_CFC_ (* Continuous Function Chart, elements in execution order *)
#0 ABS(SCHU_P2_2_YA3_RASSOG)
#1 GT(#0, SCHU_P2_2_YA3_UST_RAS_TEMP)
#2 ABS(SCHU_P2_2_YA3_RASSOG_POL)
#3 GT(#2, SCHU_P2_2_YA3_UST_RAS_POL)
#4 OR(#1, #3)
#5 AND(SCHU_P2_2_UST_LETO, SCHU_P2_2_UST_RE_RABOTA, #4)
#6 INT_TO_TIME(SCHU_P2_2_YA3_ZADER_OTK)
#7 MUL(#6, 1000)
#8 TON_YA3_Zakl:TON(IN: #5, PT: #7)
#9 OR(#8.Q, YA3_AO_OTKAZ, YA3_OTKAZ)
#10 AND(SCHU_P2_2_UE2_T_DOST, SCHU_P2_2_SA5_DI5_A, #9)
#11 SR_YA3_Otk:SR(SET1: #10, RESET: SCHU_P2_2_SB)
#12 SCHU_P2_2_Z_YA3_OTKAZ <= #11.Q1
_END_CFC_
(* the same logic as Structured Text *)
TON_YA3_Zakl(IN := SCHU_P2_2_UST_LETO AND SCHU_P2_2_UST_RE_RABOTA AND ((ABS(SCHU_P2_2_YA3_RASSOG) > SCHU_P2_2_YA3_UST_RAS_TEMP) OR (ABS(SCHU_P2_2_YA3_RASSOG_POL) > SCHU_P2_2_YA3_UST_RAS_POL)), PT := INT_TO_TIME(SCHU_P2_2_YA3_ZADER_OTK) * 1000);
SR_YA3_Otk(SET1 := SCHU_P2_2_UE2_T_DOST AND SCHU_P2_2_SA5_DI5_A AND (TON_YA3_Zakl.Q OR YA3_AO_OTKAZ OR YA3_OTKAZ), RESET := SCHU_P2_2_SB);
SCHU_P2_2_Z_YA3_OTKAZ := SR_YA3_Otk.Q1;
END_PROGRAM

(* POU TZBiS/TZB/Z_YA4_Otk, CFC *)
PROGRAM Z_YA4_Otk
VAR
	RS_YA4_OTKZ: SR;

	UE3_ZADER: TON;
	SCHU_P2_2_YA4_AO4ER: TON;
	F_trig_ai: F_TRIG;
	TON_YA4: TON;
	YA4_ZADER_POL: TON;
	YA4_ZADER_TEMP: TON;
END_VAR
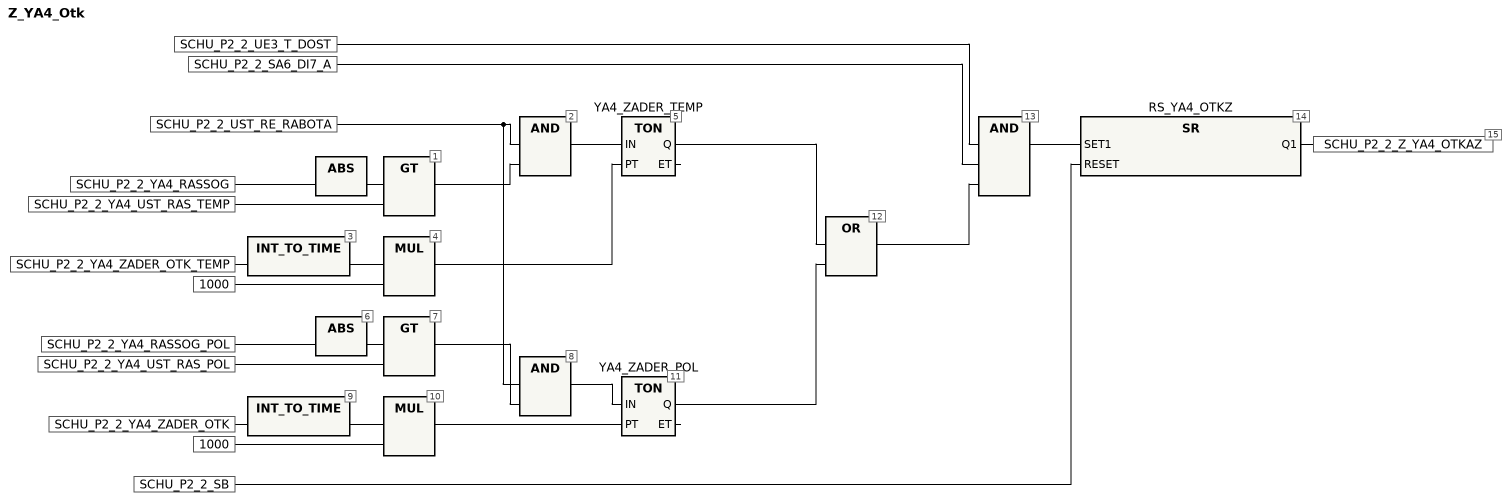
_CFC_ (* Continuous Function Chart, elements in execution order *)
#0 ABS(SCHU_P2_2_YA4_RASSOG)
#1 GT(#0, SCHU_P2_2_YA4_UST_RAS_TEMP)
#2 AND(SCHU_P2_2_UST_RE_RABOTA, #1)
#3 INT_TO_TIME(SCHU_P2_2_YA4_ZADER_OTK_TEMP)
#4 MUL(#3, 1000)
#5 YA4_ZADER_TEMP:TON(IN: #2, PT: #4)
#6 ABS(SCHU_P2_2_YA4_RASSOG_POL)
#7 GT(#6, SCHU_P2_2_YA4_UST_RAS_POL)
#8 AND(SCHU_P2_2_UST_RE_RABOTA, #7)
#9 INT_TO_TIME(SCHU_P2_2_YA4_ZADER_OTK)
#10 MUL(#9, 1000)
#11 YA4_ZADER_POL:TON(IN: #8, PT: #10)
#12 OR(#5.Q, #11.Q)
#13 AND(SCHU_P2_2_UE3_T_DOST, SCHU_P2_2_SA6_DI7_A, #12)
#14 RS_YA4_OTKZ:SR(SET1: #13, RESET: SCHU_P2_2_SB)
#15 SCHU_P2_2_Z_YA4_OTKAZ <= #14.Q1
_END_CFC_
(* the same logic as Structured Text *)
YA4_ZADER_TEMP(IN := SCHU_P2_2_UST_RE_RABOTA AND (ABS(SCHU_P2_2_YA4_RASSOG) > SCHU_P2_2_YA4_UST_RAS_TEMP), PT := INT_TO_TIME(SCHU_P2_2_YA4_ZADER_OTK_TEMP) * 1000);
YA4_ZADER_POL(IN := SCHU_P2_2_UST_RE_RABOTA AND (ABS(SCHU_P2_2_YA4_RASSOG_POL) > SCHU_P2_2_YA4_UST_RAS_POL), PT := INT_TO_TIME(SCHU_P2_2_YA4_ZADER_OTK) * 1000);
RS_YA4_OTKZ(SET1 := SCHU_P2_2_UE3_T_DOST AND SCHU_P2_2_SA6_DI7_A AND (YA4_ZADER_TEMP.Q OR YA4_ZADER_POL.Q), RESET := SCHU_P2_2_SB);
SCHU_P2_2_Z_YA4_OTKAZ := RS_YA4_OTKZ.Q1;
END_PROGRAM

(* POU TZBiS/TZB/Z_Zam, CFC *)
PROGRAM Z_Zam
VAR
	RT_VKL: R_TRIG;
	SR_ZAM: SR;
	TON_VKL: TON;
	TP_VKL: TON;
	FT_TP_VKL: F_TRIG;
	SR_TS: SR;
END_VAR
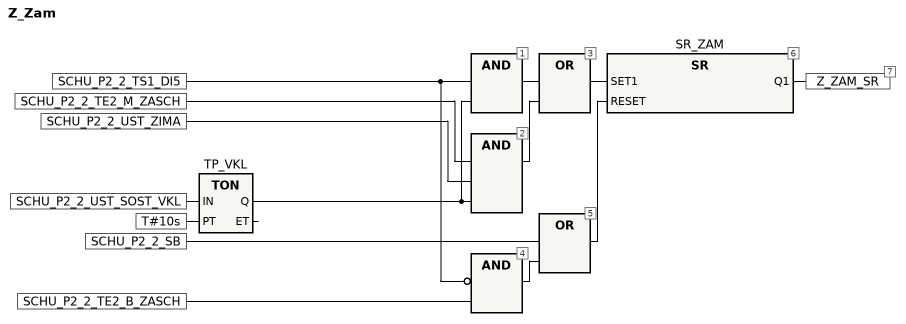
_CFC_ (* Continuous Function Chart, elements in execution order *)
#0 TP_VKL:TON(IN: SCHU_P2_2_UST_SOST_VKL, PT: T#10s)
#1 AND(SCHU_P2_2_TS1_DI5, #0.Q)
#2 AND(SCHU_P2_2_TE2_M_ZASCH, SCHU_P2_2_UST_ZIMA, #0.Q)
#3 OR(#1, #2)
#4 AND(NOT SCHU_P2_2_TS1_DI5, SCHU_P2_2_TE2_B_ZASCH)
#5 OR(SCHU_P2_2_SB, #4)
#6 SR_ZAM:SR(SET1: #3, RESET: #5)
#7 Z_ZAM_SR <= #6.Q1
_END_CFC_
(* the same logic as Structured Text *)
TP_VKL(IN := SCHU_P2_2_UST_SOST_VKL, PT := T#10s);
SR_ZAM(SET1 := (SCHU_P2_2_TS1_DI5 AND TP_VKL.Q) OR (SCHU_P2_2_TE2_M_ZASCH AND SCHU_P2_2_UST_ZIMA AND TP_VKL.Q), RESET := SCHU_P2_2_SB OR (NOT SCHU_P2_2_TS1_DI5 AND SCHU_P2_2_TE2_B_ZASCH));
Z_ZAM_SR := SR_ZAM.Q1;
END_PROGRAM

(* POU TZBiS/TZB/Z_Dlit_Ster_Reg, CFC *)
	PROGRAM Z_Dlit_Ster_Reg
VAR
	SR_HZ20S60: SR;
	LT_HZm20: ISTOK_LT;
	TON_HZm20: TON;
END_VAR
VAR (* helpers for the ST form of the networks *)
	_t19 : BOOL;
END_VAR
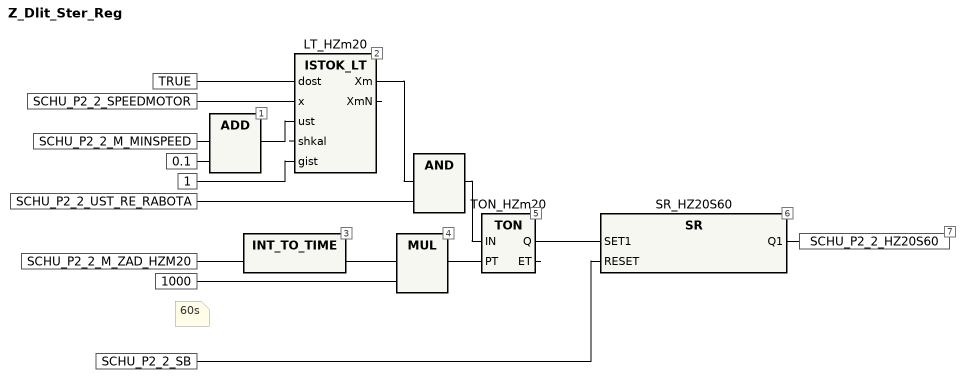
_CFC_ (* Continuous Function Chart, elements in execution order *)
(* 60s *)
#0 AND(#2.Xm, SCHU_P2_2_UST_RE_RABOTA)
#1 ADD(SCHU_P2_2_M_MINSPEED, 0.1)
#2 LT_HZm20:ISTOK_LT(dost: TRUE, x: SCHU_P2_2_SPEEDMOTOR, ust: #1, shkal: -, gist: 1)
#3 INT_TO_TIME(SCHU_P2_2_M_ZAD_HZM20)
#4 MUL(#3, 1000)
#5 TON_HZm20:TON(IN: #0, PT: #4)
#6 SR_HZ20S60:SR(SET1: #5.Q, RESET: SCHU_P2_2_SB)
#7 SCHU_P2_2_HZ20S60 <= #6.Q1
_END_CFC_
(* the same logic as Structured Text *)
(* 60s *)
_t19 := LT_HZm20.Xm AND SCHU_P2_2_UST_RE_RABOTA;
LT_HZm20(dost := TRUE, x := SCHU_P2_2_SPEEDMOTOR, ust := SCHU_P2_2_M_MINSPEED + 0.1, gist := 1);
TON_HZm20(IN := _t19, PT := INT_TO_TIME(SCHU_P2_2_M_ZAD_HZM20) * 1000);
SR_HZ20S60(SET1 := TON_HZm20.Q, RESET := SCHU_P2_2_SB);
SCHU_P2_2_HZ20S60 := SR_HZ20S60.Q1;
END_PROGRAM

(* POU TZBiS/TZB/Z_ALL, CFC *)
PROGRAM Z_ALL
VAR
	SR_Z_all: SR;
END_VAR
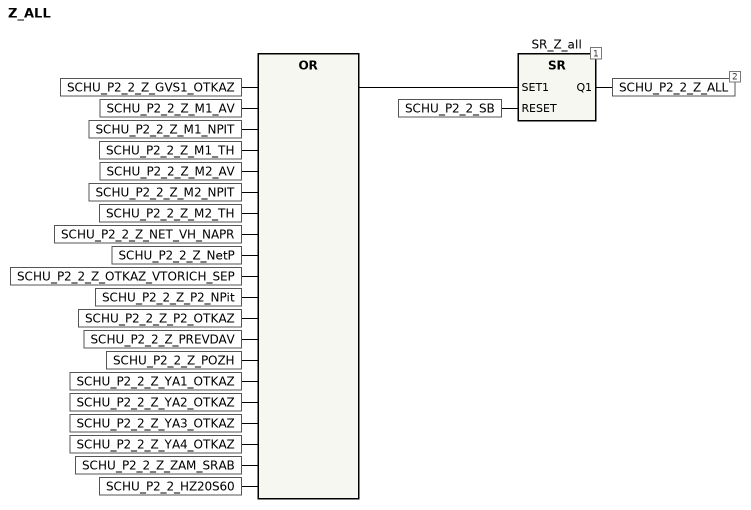
_CFC_ (* Continuous Function Chart, elements in execution order *)
#0 OR(SCHU_P2_2_Z_GVS1_OTKAZ, SCHU_P2_2_Z_M1_AV, SCHU_P2_2_Z_M1_NPIT, SCHU_P2_2_Z_M1_TH, SCHU_P2_2_Z_M2_AV, SCHU_P2_2_Z_M2_NPIT, SCHU_P2_2_Z_M2_TH, SCHU_P2_2_Z_NET_VH_NAPR, SCHU_P2_2_Z_NetP, SCHU_P2_2_Z_OTKAZ_VTORICH_SEP, SCHU_P2_2_Z_P2_NPit, SCHU_P2_2_Z_P2_OTKAZ, SCHU_P2_2_Z_PREVDAV, SCHU_P2_2_Z_POZH, SCHU_P2_2_Z_YA1_OTKAZ, SCHU_P2_2_Z_YA2_OTKAZ, SCHU_P2_2_Z_YA3_OTKAZ, SCHU_P2_2_Z_YA4_OTKAZ, SCHU_P2_2_Z_ZAM_SRAB, SCHU_P2_2_HZ20S60)
#1 SR_Z_all:SR(SET1: #0, RESET: SCHU_P2_2_SB)
#2 SCHU_P2_2_Z_ALL <= #1.Q1
_END_CFC_
(* the same logic as Structured Text *)
SR_Z_all(SET1 := SCHU_P2_2_Z_GVS1_OTKAZ OR SCHU_P2_2_Z_M1_AV OR SCHU_P2_2_Z_M1_NPIT OR SCHU_P2_2_Z_M1_TH OR SCHU_P2_2_Z_M2_AV OR SCHU_P2_2_Z_M2_NPIT OR SCHU_P2_2_Z_M2_TH OR SCHU_P2_2_Z_NET_VH_NAPR OR SCHU_P2_2_Z_NetP OR SCHU_P2_2_Z_OTKAZ_VTORICH_SEP OR SCHU_P2_2_Z_P2_NPit OR SCHU_P2_2_Z_P2_OTKAZ OR SCHU_P2_2_Z_PREVDAV OR SCHU_P2_2_Z_POZH OR SCHU_P2_2_Z_YA1_OTKAZ OR SCHU_P2_2_Z_YA2_OTKAZ OR SCHU_P2_2_Z_YA3_OTKAZ OR SCHU_P2_2_Z_YA4_OTKAZ OR SCHU_P2_2_Z_ZAM_SRAB OR SCHU_P2_2_HZ20S60, RESET := SCHU_P2_2_SB);
SCHU_P2_2_Z_ALL := SR_Z_all.Q1;
END_PROGRAM

(* POU Regim/ALL_Regim, CFC *)
PROGRAM ALL_Regim
VAR
END_VAR
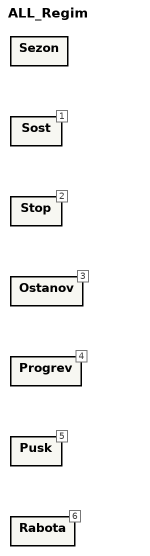
_CFC_ (* Continuous Function Chart, elements in execution order *)
#0 Sezon()
#1 Sost()
#2 Stop()
#3 Ostanov()
#4 Progrev()
#5 Pusk()
#6 Rabota()
_END_CFC_
(* the same logic as Structured Text *)
Sezon();
Sost();
Stop();
Ostanov();
Progrev();
Pusk();
Rabota();
END_PROGRAM

(* POU Regim/Sezon, CFC *)
PROGRAM Sezon
VAR
	RS_Sezon: RS;
	RT_Zima: R_TRIG;
	RT_Leto: R_TRIG;
	RT_Auto: R_TRIG;
	RS_Auto: RS;
	RT_T: R_TRIG;
END_VAR
VAR (* helpers for the ST form of the networks *)
	_t72 : BOOL;
END_VAR
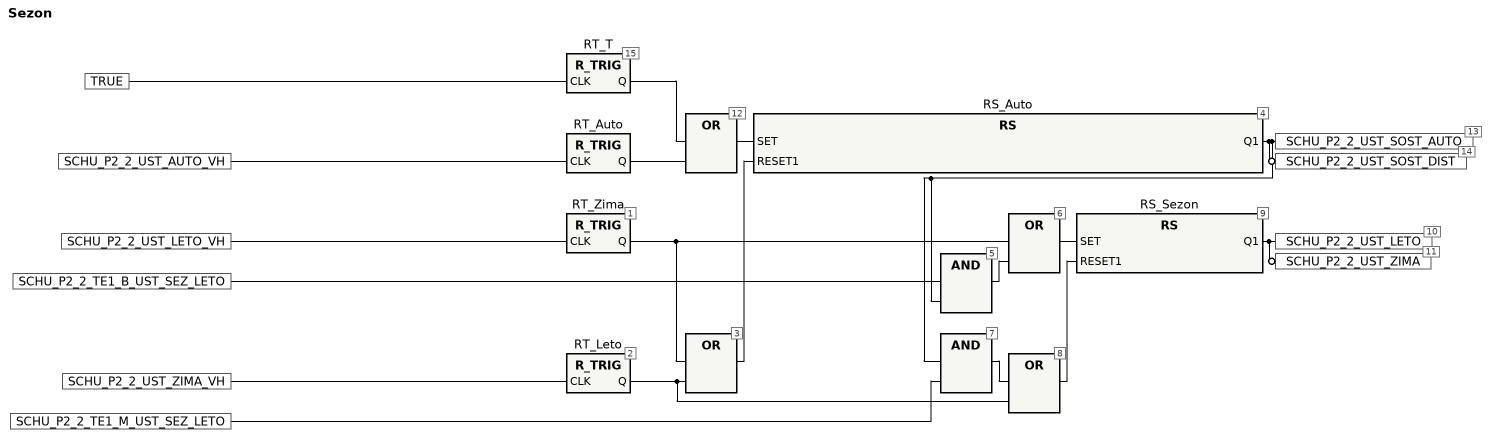
